TEXTLIST DimmingCurve
  0 = 'Standard'
  1 = 'Linear'
  255 = 'Unknown'
   = ''
END_TEXTLIST

(* stored: Version 1.1.0.1, ProductVersion 3.1.4024.12
   TextList DimmingCurve: Id {c2548d79-8137-4c31-b64d-242d60780c97} *)
